Universal Robots PolyScope program: SocketDemo.urp

Program SocketDemo (installation=default directory=/programs/Demos createdIn=5.9.1.1031110 lastSavedIn=5.11.6.1010389 robotSerialNumber=20205001585)
Calibrated DH parameters: a=[-0.000008, -0.183028, -0.487575, 0.000076, -0.000024, 0]; d=[0.180652, -404.494359, 176.775055, 227.893146, 0.119782, 0.115539]; alpha=[1.570008, -0.001443, -0.001307, 1.569929, -1.569524, 0]; deltaTheta=[0, 1.266984, 5.564204, -0.548006, 0, 0]
Robot Program (runOnlyOnce=false)
  'Host IP needs to match the static IP of the host PC (not the robot)'
  host_ip := "10.104.5.232"
  host_sock_open := socket_open(host_ip,30000,"host_socket")
  'A small delay may be needed after opening socket and sending data'
  Wait Sleep waitTime=0.5
  If host_sock_open ≟ True
    Script: socket_send_string("hello","host_socket")
    Script: socket_send_line("world","host_socket")
  Halt
